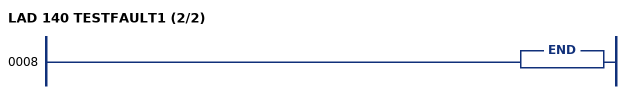
% Rung: 8 %
SOR END EOR

LADDER 141 "INS1FIX1"
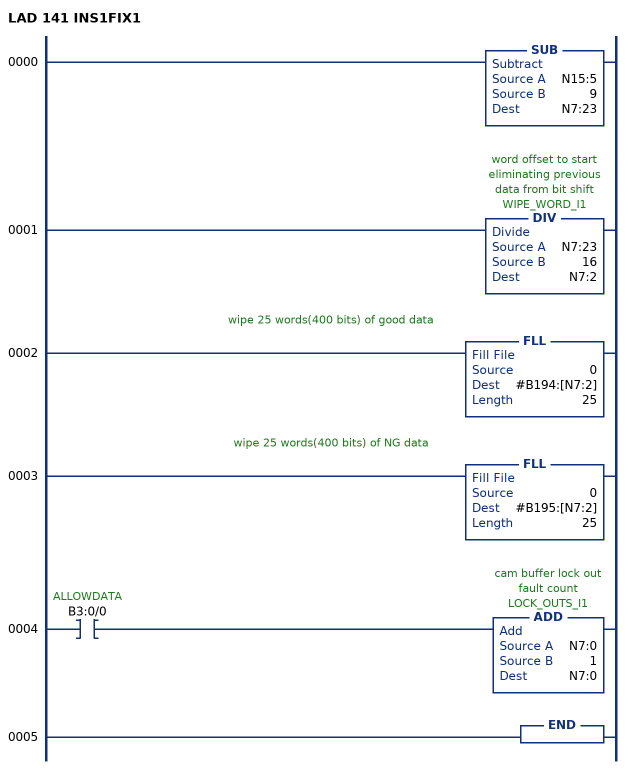
% Rung: 0 %
SOR SUB N15:5 9 N7:23 EOR
%   N15:5  INS_1_TRIG_LOC %
% Rung: 1 %
SOR DIV N7:23 16 N7:2 EOR
%   N7:2  WIPE_WORD_I1  "word offset to start eliminating previous data from bit shift" %
% Rung: 2 %
% wipe 25 words(400 bits) of good data %
SOR FLL 0 #B194:[N7:2] 25 EOR
%   N7:2  WIPE_WORD_I1  "word offset to start eliminating previous data from bit shift" %
% Rung: 3 %
% wipe 25 words(400 bits) of NG data %
SOR FLL 0 #B195:[N7:2] 25 EOR
%   N7:2  WIPE_WORD_I1  "word offset to start eliminating previous data from bit shift" %
% Rung: 4 %
SOR XIC B3:0/0 ADD N7:0 1 N7:0 EOR
%   B3:0/0  ALLOWDATA %
%   N7:0  LOCK_OUTS_I1  "cam buffer lock out fault count" %
% Rung: 5 %
SOR END EOR

LADDER 142 "INS1FIX2"
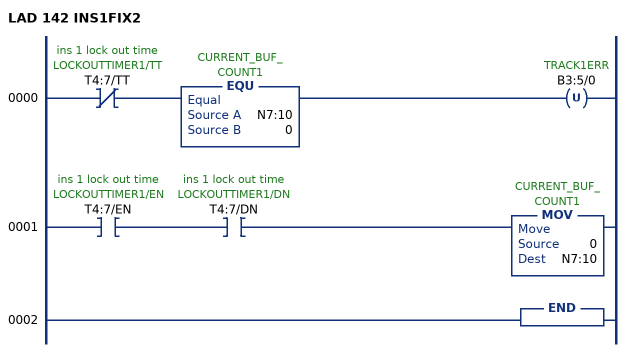
% Rung: 0 %
SOR XIO T4:7/TT EQU N7:10 0 OTU B3:5/0 EOR
%   T4:7  LOCKOUTTIMER1  "ins 1 lock out time" %
%   N7:10  CURRENT_BUF_COUNT1 %
%   B3:5/0  TRACK1ERR %
% Rung: 1 %
SOR XIC T4:7/EN XIC T4:7/DN MOV 0 N7:10 EOR
%   T4:7  LOCKOUTTIMER1  "ins 1 lock out time" %
%   N7:10  CURRENT_BUF_COUNT1 %
% Rung: 2 %
SOR END EOR

LADDER 143 "HS TRIG1"
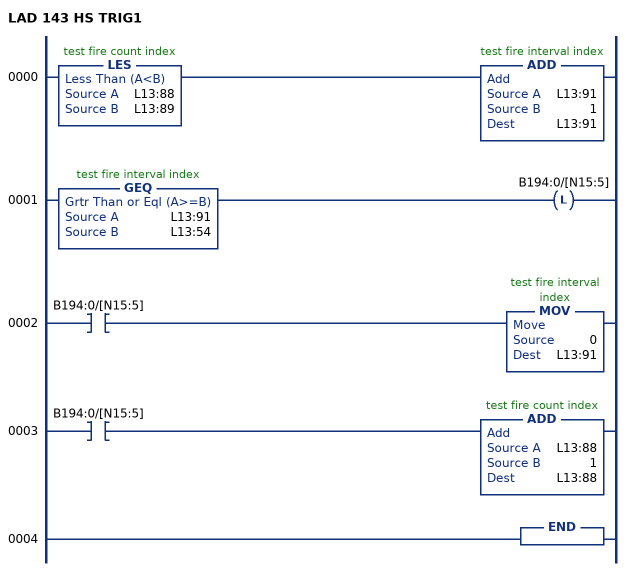
% Rung: 0 %
SOR LES L13:88 L13:89 ADD L13:91 1 L13:91 EOR
%   L13:88  "test fire count index" %
%   L13:89  "test fire count" %
%   L13:91  "test fire interval index" %
% Rung: 1 %
SOR GEQ L13:91 L13:54 OTL B194:0/[N15:5] EOR
%   L13:91  "test fire interval index" %
%   L13:54  "test fire interval" %
%   B194:0  BOT_GOOD_FILE %
%   N15:5  INS_1_TRIG_LOC %
% Rung: 2 %
SOR XIC B194:0/[N15:5] MOV 0 L13:91 EOR
%   B194:0  BOT_GOOD_FILE %
%   N15:5  INS_1_TRIG_LOC %
%   L13:91  "test fire interval index" %
% Rung: 3 %
SOR XIC B194:0/[N15:5] ADD L13:88 1 L13:88 EOR
%   B194:0  BOT_GOOD_FILE %
%   N15:5  INS_1_TRIG_LOC %
%   L13:88  "test fire count index" %
% Rung: 4 %
SOR END EOR

LADDER 145 "INS2"
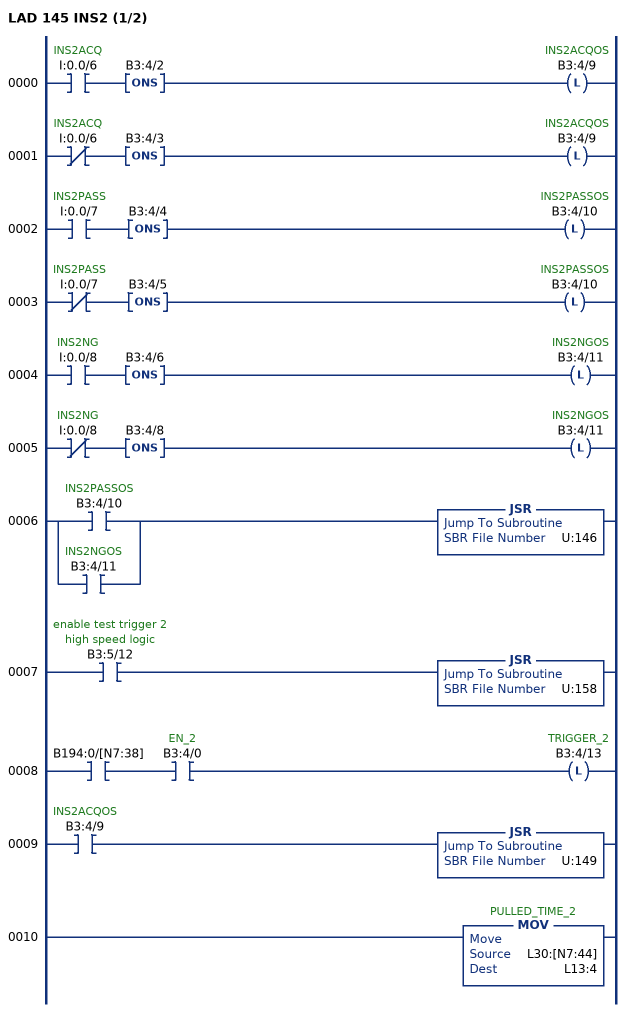
% Rung: 0 %
SOR XIC I:0.0/6 ONS B3:4/2 OTL B3:4/9 EOR
%   I:0.0/6  INS2ACQ %
%   B3:4/9  INS2ACQOS %
% Rung: 1 %
SOR XIO I:0.0/6 ONS B3:4/3 OTL B3:4/9 EOR
%   I:0.0/6  INS2ACQ %
%   B3:4/9  INS2ACQOS %
% Rung: 2 %
SOR XIC I:0.0/7 ONS B3:4/4 OTL B3:4/10 EOR
%   I:0.0/7  INS2PASS %
%   B3:4/10  INS2PASSOS %
% Rung: 3 %
SOR XIO I:0.0/7 ONS B3:4/5 OTL B3:4/10 EOR
%   I:0.0/7  INS2PASS %
%   B3:4/10  INS2PASSOS %
% Rung: 4 %
SOR XIC I:0.0/8 ONS B3:4/6 OTL B3:4/11 EOR
%   I:0.0/8  INS2NG %
%   B3:4/11  INS2NGOS %
% Rung: 5 %
SOR XIO I:0.0/8 ONS B3:4/8 OTL B3:4/11 EOR
%   I:0.0/8  INS2NG %
%   B3:4/11  INS2NGOS %
% Rung: 6 %
SOR BST XIC B3:4/10 NXB XIC B3:4/11 BND JSR U:146 EOR
%   B3:4/10  INS2PASSOS %
%   B3:4/11  INS2NGOS %
% Rung: 7 %
SOR XIC B3:5/12 JSR U:158 EOR
%   B3:5/12  "enable test trigger 2 high speed logic" %
% Rung: 8 %
SOR XIC B194:0/[N7:38] XIC B3:4/0 OTL B3:4/13 EOR
%   B194:0  BOT_GOOD_FILE %
%   N7:38  INS_2_TRIG_LOC %
%   B3:4/0  EN_2 %
%   B3:4/13  TRIGGER_2 %
% Rung: 9 %
SOR XIC B3:4/9 JSR U:149 EOR
%   B3:4/9  INS2ACQOS %
% Rung: 10 %
SOR MOV L30:[N7:44] L13:4 EOR
%   N7:44  OLDEST_PART_INDEX2 %
%   L13:4  PULLED_TIME_2 %

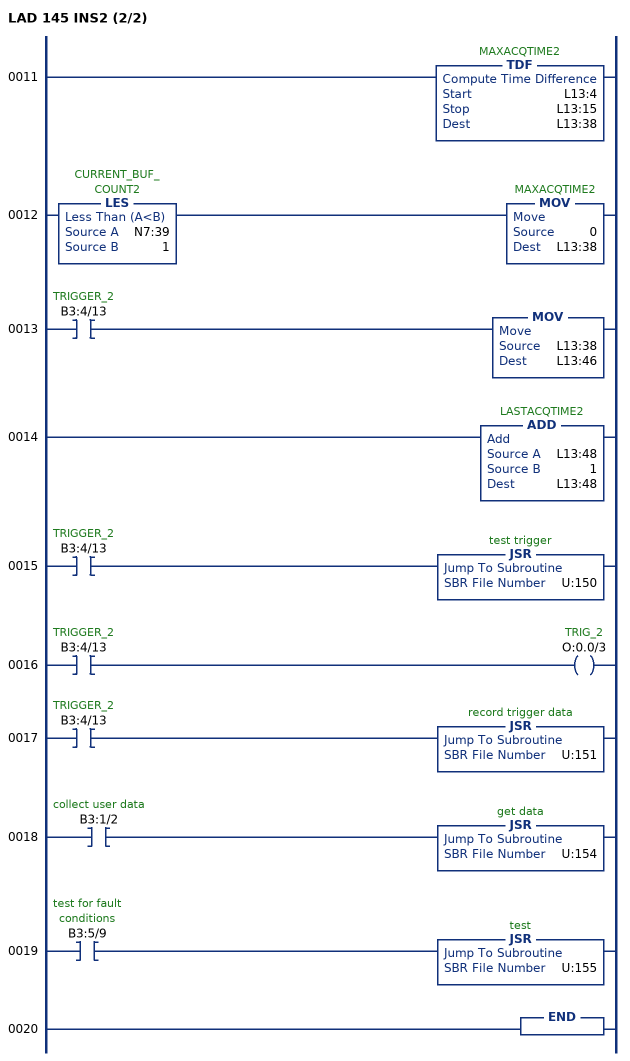
% Rung: 11 %
SOR TDF L13:4 L13:15 L13:38 EOR
%   L13:4  PULLED_TIME_2 %
%   L13:15  BOT_TIME %
%   L13:38  MAXACQTIME2 %
% Rung: 12 %
SOR LES N7:39 1 MOV 0 L13:38 EOR
%   N7:39  CURRENT_BUF_COUNT2 %
%   L13:38  MAXACQTIME2 %
% Rung: 13 %
SOR XIC B3:4/13 MOV L13:38 L13:46 EOR
%   B3:4/13  TRIGGER_2 %
%   L13:38  MAXACQTIME2 %
% Rung: 14 %
SOR ADD L13:48 1 L13:48 EOR
%   L13:48  LASTACQTIME2 %
% Rung: 15 %
SOR XIC B3:4/13 JSR U:150 EOR
%   B3:4/13  TRIGGER_2 %
%   U:150  "test trigger" %
% Rung: 16 %
SOR XIC B3:4/13 OTE O:0.0/3 EOR
%   B3:4/13  TRIGGER_2 %
%   O:0.0/3  TRIG_2 %
% Rung: 17 %
SOR XIC B3:4/13 JSR U:151 EOR
%   B3:4/13  TRIGGER_2 %
%   U:151  "record trigger data" %
% Rung: 18 %
SOR XIC B3:1/2 JSR U:154 EOR
%   B3:1/2  "collect user data" %
%   U:154  "get data" %
% Rung: 19 %
SOR XIC B3:5/9 JSR U:155 EOR
%   B3:5/9  "test for fault conditions" %
%   U:155  "test" %
% Rung: 20 %
SOR END EOR

LADDER 146 "INS2RESULT"
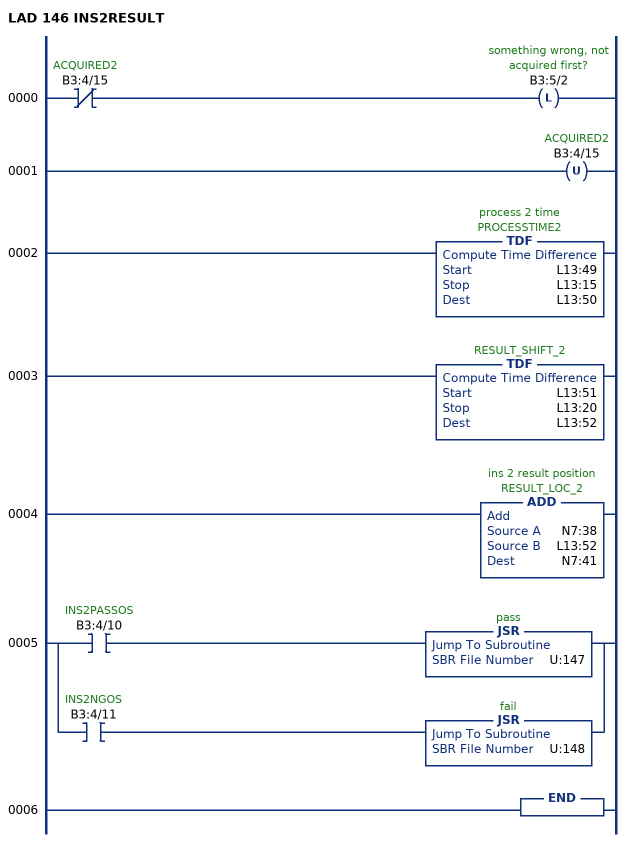
% Rung: 0 %
SOR XIO B3:4/15 OTL B3:5/2 EOR
%   B3:4/15  ACQUIRED2 %
%   B3:5/2  "something wrong, not acquired first?" %
% Rung: 1 %
SOR OTU B3:4/15 EOR
%   B3:4/15  ACQUIRED2 %
% Rung: 2 %
SOR TDF L13:49 L13:15 L13:50 EOR
%   L13:49  TIMEOFACQ2  "the time of the last acquire" %
%   L13:15  BOT_TIME %
%   L13:50  PROCESSTIME2  "process 2 time" %
% Rung: 3 %
SOR TDF L13:51 L13:20 L13:52 EOR
%   L13:51  PROCESS_START_POS_2 %
%   L13:20  BOT_POSITION %
%   L13:52  RESULT_SHIFT_2 %
% Rung: 4 %
SOR ADD N7:38 L13:52 N7:41 EOR
%   N7:38  INS_2_TRIG_LOC %
%   L13:52  RESULT_SHIFT_2 %
%   N7:41  RESULT_LOC_2  "ins 2 result position" %
% Rung: 5 %
SOR BST XIC B3:4/10 JSR U:147 NXB XIC B3:4/11 JSR U:148 BND EOR
%   B3:4/10  INS2PASSOS %
%   U:147  "pass" %
%   B3:4/11  INS2NGOS %
%   U:148  "fail" %
% Rung: 6 %
SOR END EOR

LADDER 147 "INS2PASS"
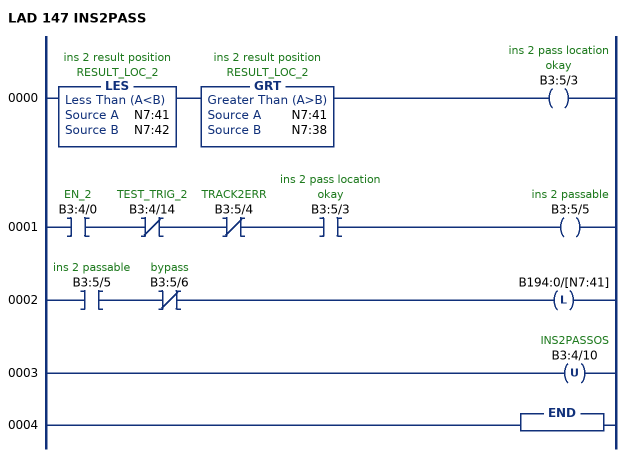
% Rung: 0 %
SOR LES N7:41 N7:42 GRT N7:41 N7:38 OTE B3:5/3 EOR
%   N7:41  RESULT_LOC_2  "ins 2 result position" %
%   N7:42  MAXRSTLOC2 %
%   N7:38  INS_2_TRIG_LOC %
%   B3:5/3  "ins 2 pass location okay" %
% Rung: 1 %
SOR XIC B3:4/0 XIO B3:4/14 XIO B3:5/4 XIC B3:5/3 OTE B3:5/5 EOR
%   B3:4/0  EN_2 %
%   B3:4/14  TEST_TRIG_2 %
%   B3:5/4  TRACK2ERR %
%   B3:5/3  "ins 2 pass location okay" %
%   B3:5/5  "ins 2 passable" %
% Rung: 2 %
SOR XIC B3:5/5 XIO B3:5/6 OTL B194:0/[N7:41] EOR
%   B3:5/5  "ins 2 passable" %
%   B3:5/6  "bypass" %
%   B194:0  BOT_GOOD_FILE %
%   N7:41  RESULT_LOC_2  "ins 2 result position" %
% Rung: 3 %
SOR OTU B3:4/10 EOR
%   B3:4/10  INS2PASSOS %
% Rung: 4 %
SOR END EOR

LADDER 148 "INS2FAIL"
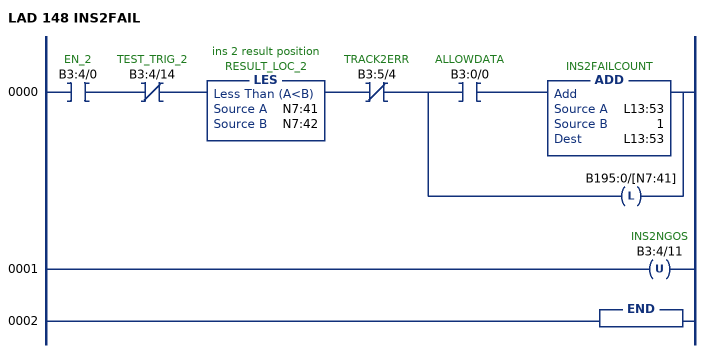
% Rung: 0 %
SOR XIC B3:4/0 XIO B3:4/14 LES N7:41 N7:42 XIO B3:5/4 BST XIC B3:0/0 ADD L13:53 1 L13:53 NXB OTL B195:0/[N7:41] BND EOR
%   B3:4/0  EN_2 %
%   B3:4/14  TEST_TRIG_2 %
%   N7:41  RESULT_LOC_2  "ins 2 result position" %
%   N7:42  MAXRSTLOC2 %
%   B3:5/4  TRACK2ERR %
%   B3:0/0  ALLOWDATA %
%   L13:53  INS2FAILCOUNT %
%   B195:0  BOT_NG_FILE %
% Rung: 1 %
SOR OTU B3:4/11 EOR
%   B3:4/11  INS2NGOS %
% Rung: 2 %
SOR END EOR

LADDER 149 "INS2ACQ"
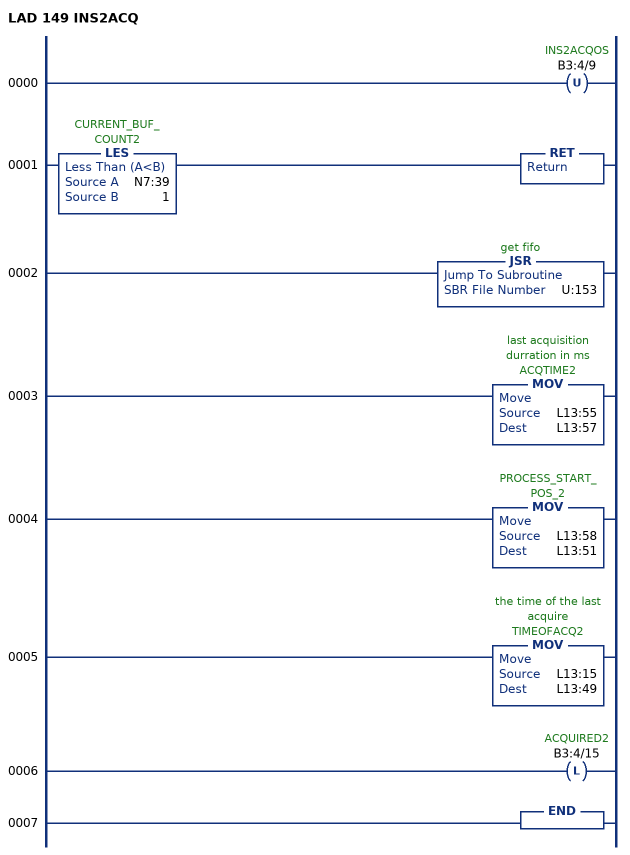
% Rung: 0 %
SOR OTU B3:4/9 EOR
%   B3:4/9  INS2ACQOS %
% Rung: 1 %
SOR LES N7:39 1 RET EOR
%   N7:39  CURRENT_BUF_COUNT2 %
% Rung: 2 %
SOR JSR U:153 EOR
%   U:153  "get fifo" %
% Rung: 3 %
SOR MOV L13:55 L13:57 EOR
%   L13:55  TIME_SPAN2 %
%   L13:57  ACQTIME2  "last acquisition durration in ms" %
% Rung: 4 %
SOR MOV L13:58 L13:51 EOR
%   L13:58  PULLED_POSITION2 %
%   L13:51  PROCESS_START_POS_2 %
% Rung: 5 %
SOR MOV L13:15 L13:49 EOR
%   L13:15  BOT_TIME %
%   L13:49  TIMEOFACQ2  "the time of the last acquire" %
% Rung: 6 %
SOR OTL B3:4/15 EOR
%   B3:4/15  ACQUIRED2 %
% Rung: 7 %
SOR END EOR

LADDER 150 "Q2TIMETEST"
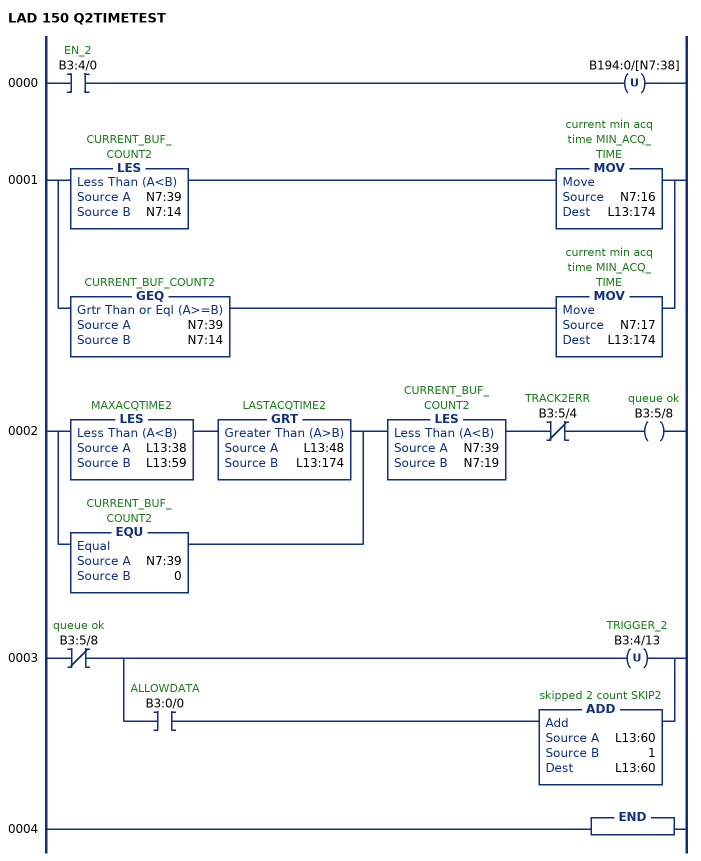
% Rung: 0 %
SOR XIC B3:4/0 OTU B194:0/[N7:38] EOR
%   B3:4/0  EN_2 %
%   B194:0  BOT_GOOD_FILE %
%   N7:38  INS_2_TRIG_LOC %
% Rung: 1 %
SOR BST LES N7:39 N7:14 MOV N7:16 L13:174 NXB GEQ N7:39 N7:14 MOV N7:17 L13:174 BND EOR
%   N7:39  CURRENT_BUF_COUNT2 %
%   N7:14  "Max high speed buffers" %
%   N7:16  "high speed acquisition time" %
%   L13:174  MIN_ACQ_TIME  "current min acq time" %
%   N7:17  "low speed acquisition time" %
% Rung: 2 %
SOR BST LES L13:38 L13:59 GRT L13:48 L13:174 NXB EQU N7:39 0 BND LES N7:39 N7:19 XIO B3:5/4 OTE B3:5/8 EOR
%   L13:38  MAXACQTIME2 %
%   L13:59  ACQTIMELIMIT2 %
%   L13:48  LASTACQTIME2 %
%   L13:174  MIN_ACQ_TIME  "current min acq time" %
%   N7:39  CURRENT_BUF_COUNT2 %
%   N7:19  MAX_BUFF  "maximum buffers" %
%   B3:5/4  TRACK2ERR %
%   B3:5/8  "queue ok" %
% Rung: 3 %
SOR XIO B3:5/8 BST OTU B3:4/13 NXB XIC B3:0/0 ADD L13:60 1 L13:60 BND EOR
%   B3:5/8  "queue ok" %
%   B3:4/13  TRIGGER_2 %
%   B3:0/0  ALLOWDATA %
%   L13:60  SKIP2  "skipped 2 count" %
% Rung: 4 %
SOR END EOR

LADDER 151 "INS2TRIG"
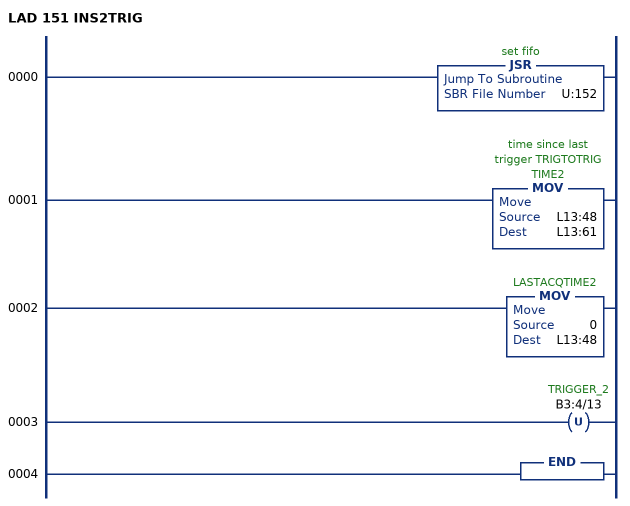
% Rung: 0 %
SOR JSR U:152 EOR
%   U:152  "set fifo" %
% Rung: 1 %
SOR MOV L13:48 L13:61 EOR
%   L13:48  LASTACQTIME2 %
%   L13:61  TRIGTOTRIGTIME2  "time since last trigger" %
% Rung: 2 %
SOR MOV 0 L13:48 EOR
%   L13:48  LASTACQTIME2 %
% Rung: 3 %
SOR OTU B3:4/13 EOR
%   B3:4/13  TRIGGER_2 %
% Rung: 4 %
SOR END EOR

LADDER 152 "FIFO2SET"
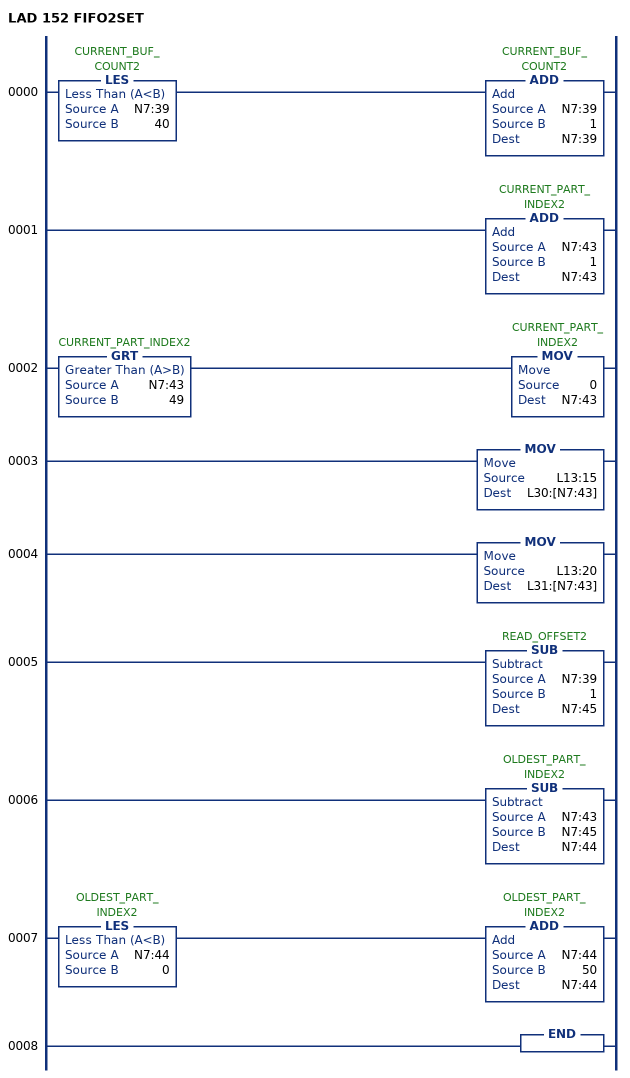
% Rung: 0 %
SOR LES N7:39 40 ADD N7:39 1 N7:39 EOR
%   N7:39  CURRENT_BUF_COUNT2 %
% Rung: 1 %
SOR ADD N7:43 1 N7:43 EOR
%   N7:43  CURRENT_PART_INDEX2 %
% Rung: 2 %
SOR GRT N7:43 49 MOV 0 N7:43 EOR
%   N7:43  CURRENT_PART_INDEX2 %
% Rung: 3 %
SOR MOV L13:15 L30:[N7:43] EOR
%   L13:15  BOT_TIME %
%   N7:43  CURRENT_PART_INDEX2 %
% Rung: 4 %
SOR MOV L13:20 L31:[N7:43] EOR
%   L13:20  BOT_POSITION %
%   N7:43  CURRENT_PART_INDEX2 %
% Rung: 5 %
SOR SUB N7:39 1 N7:45 EOR
%   N7:39  CURRENT_BUF_COUNT2 %
%   N7:45  READ_OFFSET2 %
% Rung: 6 %
SOR SUB N7:43 N7:45 N7:44 EOR
%   N7:43  CURRENT_PART_INDEX2 %
%   N7:45  READ_OFFSET2 %
%   N7:44  OLDEST_PART_INDEX2 %
% Rung: 7 %
SOR LES N7:44 0 ADD N7:44 50 N7:44 EOR
%   N7:44  OLDEST_PART_INDEX2 %
% Rung: 8 %
SOR END EOR

LADDER 153 "FIFO2GET"
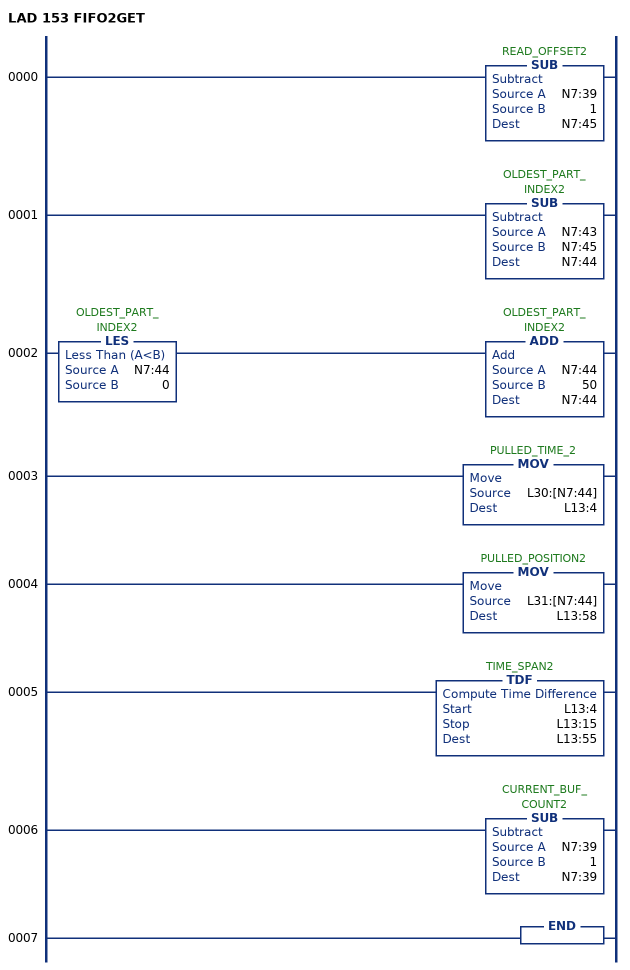
% Rung: 0 %  % edit flag set %
SOR SUB N7:39 1 N7:45 EOR
%   N7:39  CURRENT_BUF_COUNT2 %
%   N7:45  READ_OFFSET2 %
% Rung: 1 %  % edit flag set %
SOR SUB N7:43 N7:45 N7:44 EOR
%   N7:43  CURRENT_PART_INDEX2 %
%   N7:45  READ_OFFSET2 %
%   N7:44  OLDEST_PART_INDEX2 %
% Rung: 2 %
SOR LES N7:44 0 ADD N7:44 50 N7:44 EOR
%   N7:44  OLDEST_PART_INDEX2 %
% Rung: 3 %
SOR MOV L30:[N7:44] L13:4 EOR
%   N7:44  OLDEST_PART_INDEX2 %
%   L13:4  PULLED_TIME_2 %
% Rung: 4 %
SOR MOV L31:[N7:44] L13:58 EOR
%   N7:44  OLDEST_PART_INDEX2 %
%   L13:58  PULLED_POSITION2 %
% Rung: 5 %
SOR TDF L13:4 L13:15 L13:55 EOR
%   L13:4  PULLED_TIME_2 %
%   L13:15  BOT_TIME %
%   L13:55  TIME_SPAN2 %
% Rung: 6 %
SOR SUB N7:39 1 N7:39 EOR
%   N7:39  CURRENT_BUF_COUNT2 %
% Rung: 7 %
SOR END EOR

LADDER 154 "INSDATA2"    % used for analysis %
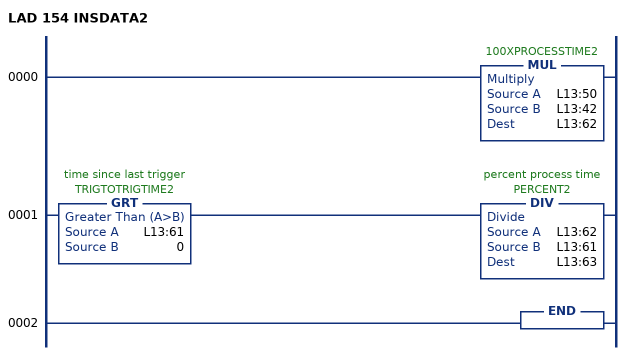
% Rung: 0 %
SOR MUL L13:50 L13:42 L13:62 EOR
%   L13:50  PROCESSTIME2  "process 2 time" %
%   L13:42  100X_MULTIPLIER %
%   L13:62  100XPROCESSTIME2 %
% Rung: 1 %
SOR GRT L13:61 0 DIV L13:62 L13:61 L13:63 EOR
%   L13:61  TRIGTOTRIGTIME2  "time since last trigger" %
%   L13:62  100XPROCESSTIME2 %
%   L13:63  PERCENT2  "percent process time" %
% Rung: 2 %
SOR END EOR

LADDER 155 "TESTFAULT2"
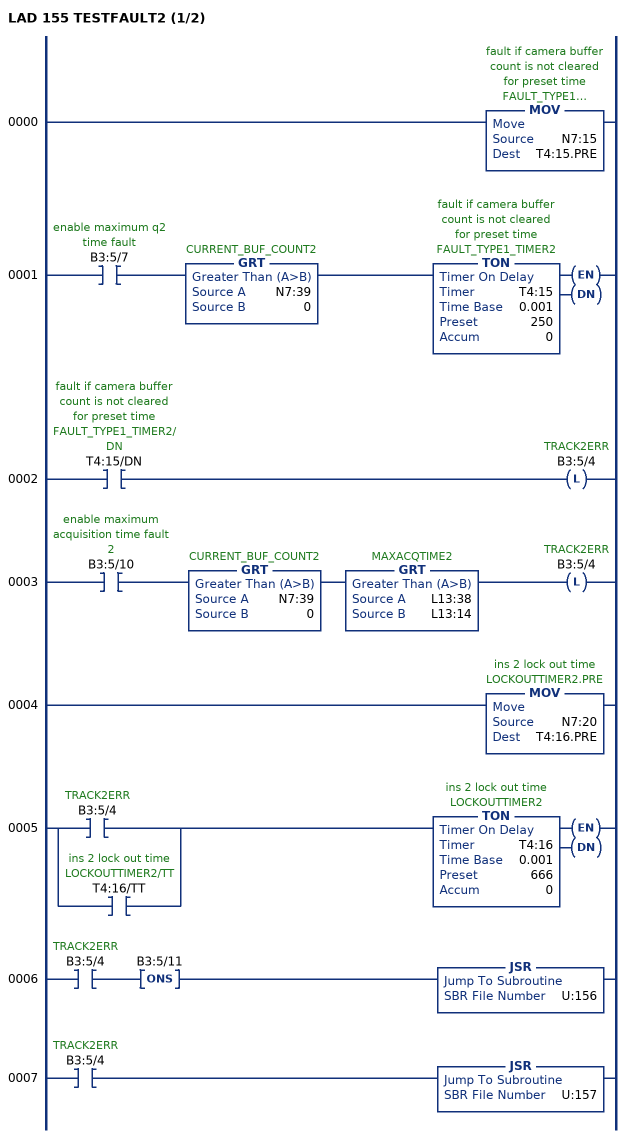
% Rung: 0 %
SOR MOV N7:15 T4:15.PRE EOR
%   N7:15  MAXQ1TMFLT  "max allowed ms time for q to be above 1 if safe fault is used" %
%   T4:15  FAULT_TYPE1_TIMER2  "fault if camera buffer count is not cleared for preset time" %
% Rung: 1 %
SOR XIC B3:5/7 GRT N7:39 0 TON T4:15 0.001 250 0 EOR
%   B3:5/7  "enable maximum q2 time fault" %
%   N7:39  CURRENT_BUF_COUNT2 %
%   T4:15  FAULT_TYPE1_TIMER2  "fault if camera buffer count is not cleared for preset time" %
% Rung: 2 %
SOR XIC T4:15/DN OTL B3:5/4 EOR
%   T4:15  FAULT_TYPE1_TIMER2  "fault if camera buffer count is not cleared for preset time" %
%   B3:5/4  TRACK2ERR %
% Rung: 3 %
SOR XIC B3:5/10 GRT N7:39 0 GRT L13:38 L13:14 OTL B3:5/4 EOR
%   B3:5/10  "enable maximum acquisition time fault 2" %
%   N7:39  CURRENT_BUF_COUNT2 %
%   L13:38  MAXACQTIME2 %
%   L13:14  LONGESTACQUIRETIME  "maximum of the longest acquire time allowed if maximum acquire time fault is enabled" %
%   B3:5/4  TRACK2ERR %
% Rung: 4 %
SOR MOV N7:20 T4:16.PRE EOR
%   N7:20  LOCKOUTTIME  "ms time setting to lock out inspection to give all pending images a chance to clear" %
%   T4:16  LOCKOUTTIMER2  "ins 2 lock out time" %
% Rung: 5 %
SOR BST XIC B3:5/4 NXB XIC T4:16/TT BND TON T4:16 0.001 666 0 EOR
%   B3:5/4  TRACK2ERR %
%   T4:16  LOCKOUTTIMER2  "ins 2 lock out time" %
% Rung: 6 %
SOR XIC B3:5/4 ONS B3:5/11 JSR U:156 EOR
%   B3:5/4  TRACK2ERR %
% Rung: 7 %
SOR XIC B3:5/4 JSR U:157 EOR
%   B3:5/4  TRACK2ERR %

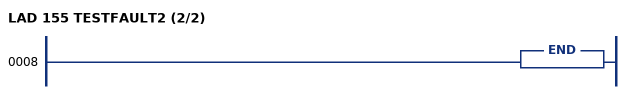
% Rung: 8 %
SOR END EOR

LADDER 156 "INS2FIX1"
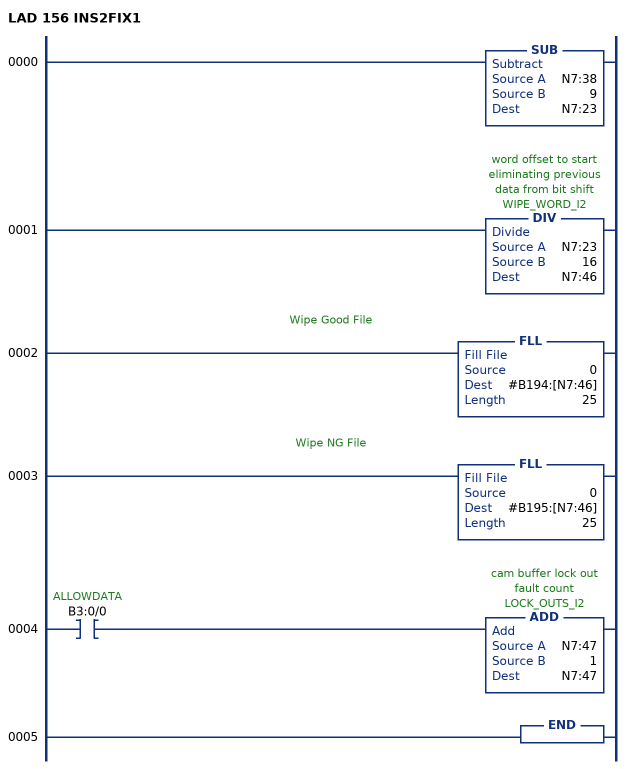
% Rung: 0 %
SOR SUB N7:38 9 N7:23 EOR
%   N7:38  INS_2_TRIG_LOC %
% Rung: 1 %
SOR DIV N7:23 16 N7:46 EOR
%   N7:46  WIPE_WORD_I2  "word offset to start eliminating previous data from bit shift" %
% Rung: 2 %
% Wipe Good File %
SOR FLL 0 #B194:[N7:46] 25 EOR
%   N7:46  WIPE_WORD_I2  "word offset to start eliminating previous data from bit shift" %
% Rung: 3 %
% Wipe NG File %
SOR FLL 0 #B195:[N7:46] 25 EOR
%   N7:46  WIPE_WORD_I2  "word offset to start eliminating previous data from bit shift" %
% Rung: 4 %
SOR XIC B3:0/0 ADD N7:47 1 N7:47 EOR
%   B3:0/0  ALLOWDATA %
%   N7:47  LOCK_OUTS_I2  "cam buffer lock out fault count" %
% Rung: 5 %
SOR END EOR

LADDER 157 "INS2FIX2"
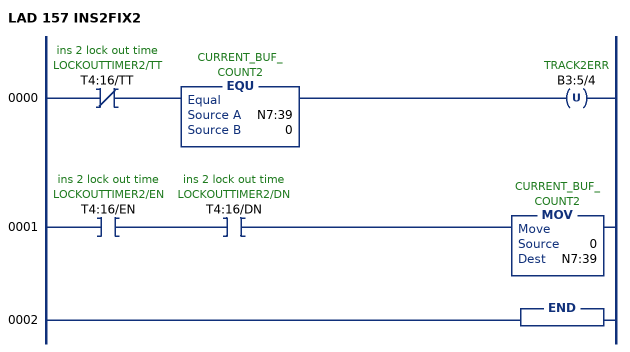
% Rung: 0 %
SOR XIO T4:16/TT EQU N7:39 0 OTU B3:5/4 EOR
%   T4:16  LOCKOUTTIMER2  "ins 2 lock out time" %
%   N7:39  CURRENT_BUF_COUNT2 %
%   B3:5/4  TRACK2ERR %
% Rung: 1 %
SOR XIC T4:16/EN XIC T4:16/DN MOV 0 N7:39 EOR
%   T4:16  LOCKOUTTIMER2  "ins 2 lock out time" %
%   N7:39  CURRENT_BUF_COUNT2 %
% Rung: 2 %
SOR END EOR

LADDER 158 "HS TRIG2"
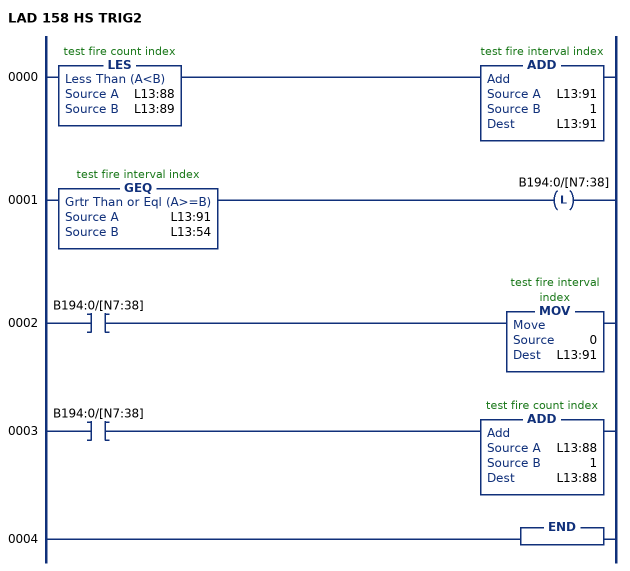
% Rung: 0 %
SOR LES L13:88 L13:89 ADD L13:91 1 L13:91 EOR
%   L13:88  "test fire count index" %
%   L13:89  "test fire count" %
%   L13:91  "test fire interval index" %
% Rung: 1 %
SOR GEQ L13:91 L13:54 OTL B194:0/[N7:38] EOR
%   L13:91  "test fire interval index" %
%   L13:54  "test fire interval" %
%   B194:0  BOT_GOOD_FILE %
%   N7:38  INS_2_TRIG_LOC %
% Rung: 2 %
SOR XIC B194:0/[N7:38] MOV 0 L13:91 EOR
%   B194:0  BOT_GOOD_FILE %
%   N7:38  INS_2_TRIG_LOC %
%   L13:91  "test fire interval index" %
% Rung: 3 %
SOR XIC B194:0/[N7:38] ADD L13:88 1 L13:88 EOR
%   B194:0  BOT_GOOD_FILE %
%   N7:38  INS_2_TRIG_LOC %
%   L13:88  "test fire count index" %
% Rung: 4 %
SOR END EOR

LADDER 200 "XFEROUT"
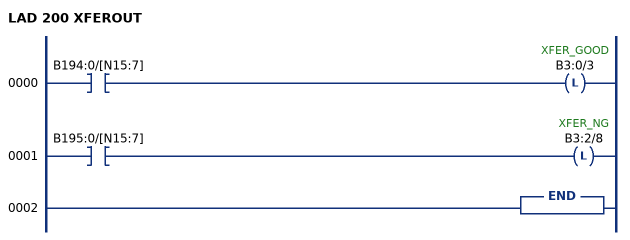
% Rung: 0 %
SOR XIC B194:0/[N15:7] OTL B3:0/3 EOR
%   B194:0  BOT_GOOD_FILE %
%   N15:7  XFER_OUT_LOC %
%   B3:0/3  XFER_GOOD %
% Rung: 1 %
SOR XIC B195:0/[N15:7] OTL B3:2/8 EOR
%   B195:0  BOT_NG_FILE %
%   N15:7  XFER_OUT_LOC %
%   B3:2/8  XFER_NG %
% Rung: 2 %
SOR END EOR

LADDER 201 "XFER GOOD"
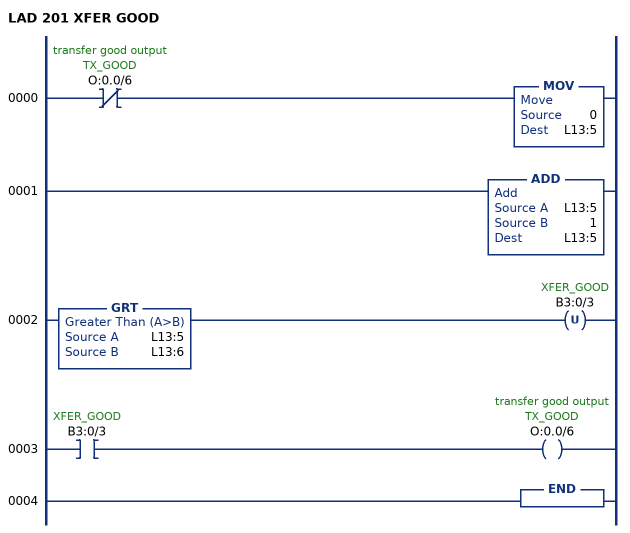
% Rung: 0 %
SOR XIO O:0.0/6 MOV 0 L13:5 EOR
%   O:0.0/6  TX_GOOD  "transfer good output" %
% Rung: 1 %
SOR ADD L13:5 1 L13:5 EOR
% Rung: 2 %
SOR GRT L13:5 L13:6 OTU B3:0/3 EOR
%   B3:0/3  XFER_GOOD %
% Rung: 3 %
SOR XIC B3:0/3 OTE O:0.0/6 EOR
%   B3:0/3  XFER_GOOD %
%   O:0.0/6  TX_GOOD  "transfer good output" %
% Rung: 4 %
SOR END EOR

LADDER 202 "XFER NG"
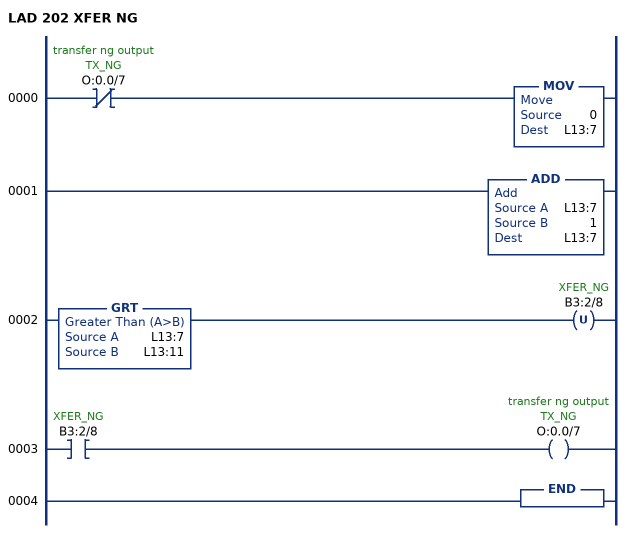
% Rung: 0 %
SOR XIO O:0.0/7 MOV 0 L13:7 EOR
%   O:0.0/7  TX_NG  "transfer ng output" %
% Rung: 1 %
SOR ADD L13:7 1 L13:7 EOR
% Rung: 2 %
SOR GRT L13:7 L13:11 OTU B3:2/8 EOR
%   B3:2/8  XFER_NG %
% Rung: 3 %
SOR XIC B3:2/8 OTE O:0.0/7 EOR
%   B3:2/8  XFER_NG %
%   O:0.0/7  TX_NG  "transfer ng output" %
% Rung: 4 %
SOR END EOR

LADDER 222 "RATE1"
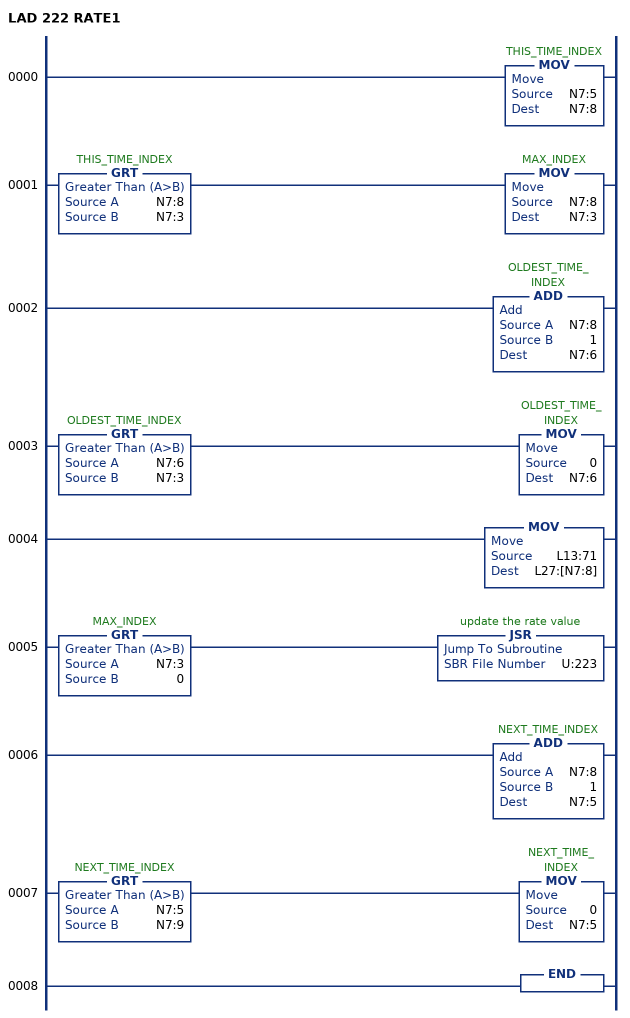
% Rung: 0 %
SOR MOV N7:5 N7:8 EOR
%   N7:5  NEXT_TIME_INDEX %
%   N7:8  THIS_TIME_INDEX %
% Rung: 1 %
SOR GRT N7:8 N7:3 MOV N7:8 N7:3 EOR
%   N7:8  THIS_TIME_INDEX %
%   N7:3  MAX_INDEX %
% Rung: 2 %
SOR ADD N7:8 1 N7:6 EOR
%   N7:8  THIS_TIME_INDEX %
%   N7:6  OLDEST_TIME_INDEX %
% Rung: 3 %
SOR GRT N7:6 N7:3 MOV 0 N7:6 EOR
%   N7:6  OLDEST_TIME_INDEX %
%   N7:3  MAX_INDEX %
% Rung: 4 %
SOR MOV L13:71 L27:[N7:8] EOR
%   L13:71  HSC_TIME %
%   N7:8  THIS_TIME_INDEX %
% Rung: 5 %
SOR GRT N7:3 0 JSR U:223 EOR
%   N7:3  MAX_INDEX %
%   U:223  "update the rate value" %
% Rung: 6 %
SOR ADD N7:8 1 N7:5 EOR
%   N7:8  THIS_TIME_INDEX %
%   N7:5  NEXT_TIME_INDEX %
% Rung: 7 %
SOR GRT N7:5 N7:9 MOV 0 N7:5 EOR
%   N7:5  NEXT_TIME_INDEX %
%   N7:9  UPPER_INDEX_LIMIT %
% Rung: 8 %
SOR END EOR

LADDER 223 "RATE2"
